          f=[0,0.0,0.0,0.0,0.0,0.0,0.0,0]
          object_location=p[0.0,0.0,0.0,0.0,0.0,0.0]
          feature_pose_to_restore_26962 = Calib_2
          movej([-1.5836804548846644, -1.5576728147319336, -1.1589980125427246, -2.3950706921019496, 1.6015324592590332, -3.158562485371725])
          # Offset in translation only.
          snapshot_position_offset[3] = 0
          snapshot_position_offset[4] = 0
          snapshot_position_offset[5] = 0
          T_camera_in_flange = p[0, 0, 0, 0, 0, 0] # enlever une fois que l'enseignement du modele sera fait en faisant un movetool avec la pose de la camera dans le repere de la flange. Pour l'instant, on suppose que la camera est situee directement sur la flange.
          tool_26962 = get_T_in_base_from_flange(T_camera_in_flange)
          tool_26962 = pose_sub(tool_26962, snapshot_position_offset)
          snapshot_position = p[-0.129407, -0.233098, 0.365602, -2.74117, -0.00825141, -0.0507442]
          textmsg("expected snapshot position : ", snapshot_position)
          diff = pose_sub(tool_26962, snapshot_position)
          textmsg("diff = ", diff)
          is_at_snapshot_position = norm([diff[0], diff[1], diff[2]]) < 0.002
          is_at_snapshot_position = is_at_snapshot_position and (norm([diff[3], diff[4], diff[5]]) < 0.005)
          textmsg("is_at_snapshot_position = ", is_at_snapshot_position)
          is_snapshot_position_offset = norm(snapshot_position_offset) != 0
          is_at_snapshot_position = is_at_snapshot_position or ignore_snapshot_position
          if not(is_at_snapshot_position):
            popup("Robot is not at Snapshot Position. Add Move instruction to Snapshot Position before Camera Locate node.. Error code: [UCC-8]", warning = False, error = True)
            halt
          end
          f_26962 = xmlrpc_server.findmodel("contextName-26962", tool_26962[0], tool_26962[1], tool_26962[2], tool_26962[3], tool_26962[4], tool_26962[5])
          cam_locate_monitor.setFindModelResult("26962", f_26962)
          canSaveImage = True
          logging_service.publish("FIND_MODEL", f_26962)
          cam_locate_monitor.setCurrentObjectIndex("26962", 0)
          # begin: URCap Program Node
          #   Source: Robotiq_Wrist_Camera, 1.10.3.5692, Robotiq Inc.
          #   Type: Boucle de la localisation de caméra
          $ 52 "Pour le ou les objets trouvés" "noBreak"
          object_teaching_location_26962 = p[-0.10858899682842695, -0.3298791170798341, 0.0013903307483954478, 2.186047489594667, -2.254339148656133, 0.01142036475668008]
          feature_teaching_location_26962 = p[-0.10858899682842695, -0.3298791170798341, 0.0013903307483954478, 2.246406672318401, 2.1857773971702463, -0.00217120647840988]
          while (not cam_locate_monitor.isCaptureNeeded("26962")):
            poseAsArray = cam_locate_monitor.getCurrentObjectPoseAsArray("26962")
            current_object_location_26962 = p[poseAsArray[0], poseAsArray[1], poseAsArray[2], poseAsArray[3], poseAsArray[4], poseAsArray[5]]
            object_location = current_object_location_26962
            f[0] = cam_locate_monitor.getNumberOfObjectsFound("26962")
            f[1] = object_location[0]
            f[2] = object_location[1]
            f[3] = object_location[2]
            f[4] = object_location[3]
            f[5] = object_location[4]
            f[6] = object_location[5]
            f[7] = cam_locate_monitor.getCurrentObjectDetectionScore("26962")
            textmsg("current_object_location = ", current_object_location_26962)
            if (norm(snapshot_position_offset) != 0):
              current_object_location_26962 = pose_add(current_object_location_26962, snapshot_position_offset)
              textmsg("current_object_location after snapshot position offset = ", current_object_location_26962)
            end
            Calib_2 = pose_trans(current_object_location_26962, pose_trans(pose_inv(object_teaching_location_26962), feature_teaching_location_26962))
            $ 53 "DéplacementL" "noBreak"
            $ 54 "approche" "noBreak"
            movel(pose_trans(Calib_1, pose_trans(p[.379088257553, .105726585325, -.047506941904, -2.247767499877, -2.191131924773, .000032734924], approche_p)), a=0.5079997256801482, v=0.4)
            $ 55 "recup" "noBreak"
            movel(pose_trans(Calib_1, pose_trans(p[.379088257553, .105726585325, -.047506941904, -2.247767499877, -2.191131924773, .000032734924], recup_p)), a=0.08, v=0.15)
            # begin: URCap Program Node
            #   Source: Robotiq_Grippers, 1.8.6.7016, Robotiq Inc.
            #   Type: Main
            $ 56 "Déplacement main55% (1)" "noBreak"
            if not(gripper_connected[0]):
              popup("Main 1 doit être connectée pour exécuter ce programme.", "Aucune connexion", False, True, True)
            end
            if not(rq_is_gripper_activated("1")):
              popup("Main 1 n’est pas activé. Accédez à l’onglet Installation > Gripper (Main) pour l’activer et exécutez à nouveau le programme.", "Non activé", False, True, True)
            end
            rq_set_pos_spd_for(140, 0, 0, "1")
            rq_wait_pos_spe_for_request(140, 0, 0, "1")
            rq_go_to("1")
            rq_wait("1")
            # end: URCap Program Node
            $ 57 "approche" "noBreak"
            movel(pose_trans(Calib_1, pose_trans(p[.379088257553, .105726585325, -.047506941904, -2.247767499877, -2.191131924773, .000032734924], approche_p)), a=0.08, v=0.15)
            $ 58 "post_prise" "noBreak"
            movel(pose_trans(Calib_1, pose_trans(p[.162610803914, -.321046559122, -.023829538781, -3.138426557699, .092719409522, -.002867798617], post_prise_p)), a=1.2, v=0.25)
            $ 59 "var_1≔ False " "noBreak"
            global var_1=  False
            $ 60 "DéplacementA" "noBreak"
            $ 61 "pro_placer" "noBreak"
            movej(get_inverse_kin(pro_placer_p, qnear=pro_placer_q), a=1.3962634015954636, v=1.3962634015954636)
            $ 62 "Placer_rebus" "noBreak"
            movej(get_inverse_kin(Placer_rebus_p, qnear=Placer_rebus_q), a=1.3962634015954636, v=1.3962634015954636)
            # begin: URCap Program Node
            #   Source: Robotiq_Grippers, 1.8.6.7016, Robotiq Inc.
            #   Type: Main
            $ 63 "Ouverture main (1)" "noBreak"
            if not(gripper_connected[0]):
              popup("Main 1 doit être connectée pour exécuter ce programme.", "Aucune connexion", False, True, True)
            end
            if not(rq_is_gripper_activated("1")):
              popup("Main 1 n’est pas activé. Accédez à l’onglet Installation > Gripper (Main) pour l’activer et exécutez à nouveau le programme.", "Non activé", False, True, True)
            end
            rq_set_pos_spd_for(0, 0, 0, "1")
            rq_wait_pos_spe_for_request(0, 0, 0, "1")
            rq_go_to("1")
            rq_wait("1")
            # end: URCap Program Node
            $ 64 "PointPassage_6" "noBreak"
            movej(get_inverse_kin(PointPassage_6_p, qnear=PointPassage_6_q), a=1.3962634015954636, v=1.3962634015954636)
            $ 65 "retour_securise" "noBreak"
            movej(get_inverse_kin(retour_securise_p, qnear=retour_securise_q), a=1.3962634015954636, v=1.3962634015954636)
            cam_locate_monitor.incrementIndex("26962")
          end
          # end: URCap Program Node
          # begin: URCap Program Node
          #   Source: Robotiq_Wrist_Camera, 1.10.3.5692, Robotiq Inc.
          #   Type: Si aucun objet n’est détecté par la caméra
          $ 66 "Si aucun objet n’est détecté" "noBreak"
          if (not cam_locate_monitor.hasFoundObjects("26962")):
            f[0] = 0
            $ 67 "'Optionnel'" "noBreak"
            # 'Optionnel'
          end
          # end: URCap Program Node
          # Restore feature pose
          Calib_2 = feature_pose_to_restore_26962

          #######VisionLocate node end########
          ###########################################

          # end: URCap Program Node
        end
      end
    end
  end
end
